{attribute 'GeneratedUsingTerminal: EP2316-0003-0016'}
{attribute addProperty BoxType "EP2316-0003-0016"}
{attribute addProperty Id "OutputAT %Q*ARRAY[0..7] OF BOOL8"}
{attribute addProperty CRC "1253840710"}
{attribute addProperty Size "8"}
TYPE DIG_Outputs_28AC1A9E :
STRUCT
	{attribute addProperty Name "Output"}
	Output AT %Q* : ARRAY[0..7] OF BOOL;
END_STRUCT
END_TYPE

(* stored: Version 1.2.0.0, ProductVersion 3.1.4024.9
   DUT DIG_Outputs_28AC1A9E: Id {80a415fb-df2b-493a-8cd9-fbe35bba182c} *)
